PROGRAM MAIN
VAR
END_VAR

Device_Diag();
EtherCAT_Diag();

END_PROGRAM

(* stored: Version 1.1.0.1, ProductVersion 3.1.4024.12
   POU MAIN: Id {43318289-7795-49fe-b0bc-d6c09020960d}, SpecialFunc None *)
